{attribute 'GeneratedUsingTerminal: EL5101-0010-0016'}
{attribute addProperty BoxType "EL5101-0010-0016"}
{attribute addProperty Id "StatusAT %I*Status_E2E79E8513Counter_valueAT %I*UINT2Latch_valueAT %I*UINT2"}
{attribute addProperty CRC "1100541755"}
{attribute addProperty Size "17"}
TYPE ENC_Status_compact_4198EF3B :
STRUCT
	{attribute addProperty Name "Status"}
	Status AT %I* : Status_E2E79E85;
	{attribute addProperty Name "Counter_value"}
	Counter_value AT %I* : UINT;
	{attribute addProperty Name "Latch_value"}
	Latch_value AT %I* : UINT;
END_STRUCT
END_TYPE

(* stored: Version 1.2.0.0, ProductVersion 3.1.4024.9
   DUT ENC_Status_compact_4198EF3B: Id {8c00abc9-6ae5-459e-8e66-a2a893cbc369} *)
